# EPICS substitutions: example/exampleApp/Db/bl0-SE-ColeParmer.substitutions
file CP-RS232_General.template
{pattern
	{ bl, ta, dn}
	{BL0F, SE, CP}
}
